FUNCTION_BLOCK FB_SignalTower
VAR_INPUT
    // TRUE: Activates the defined operation
    // FALSE: Aborts/resets the defined operation
    Enable     :BOOL := TRUE;
    LampRed    :REFERENCE TO BOOL;
    LampYellow :REFERENCE TO BOOL;
    LampGreen  :REFERENCE TO BOOL;
    Buzz       :REFERENCE TO BOOL;
	ForceCloseBuzz : BOOL;
	BuzzSwitchOnTime	:LREAL :=3000.0 ; //In Second
END_VAR

VAR_OUTPUT
    // TRUE: Operation is running
    Vaild :BOOL;
    // TRUE: Error condition reached
    Error :BOOL;
    // Error code describing error condition
    ErrorID :DINT;
END_VAR

VAR
    LampRed_Active    :BOOL;         // True :Lamp Red actived
    LampYellow_Active :BOOL;         // True :Lamp Yellow actived
    LampGreen_Active  :BOOL;         // True : Lamp Green actived
    FB_1Hz            :FB_SignalGen; // 1Hz flash signal generator
    FB_2Hz            :FB_SignalGen; // 2Hz flash signal generator
    FB_05Hz           :FB_SignalGen; // 0.5 Hz flash signal generator
    // Signal Tower controller output
    LampSingal :ST_SignalTower;
	BuzzOnTimer			:TON;

END_VAR

// Call Signal generator
A_SignalGenerator();

// 
IF Enable THEN
	LampSingal.Lamp_Red 	:= M_LampRed();
	LampSingal.Lamp_Yellow	:= M_LampYellow();
	LampSingal.Lamp_Green 	:= M_LampGreen();
	LampSingal.Buzz			:=M_Buzz(BuzzSwitchOnTime);
ELSE
	LampSingal.Lamp_Red := FALSE;
	LampSingal.Lamp_Yellow := FALSE;
	LampSingal.Lamp_Green := FALSE;
	LampSingal.Buzz := FALSE;
END_IF

LampRed := LampSingal.Lamp_Red;
LampYellow := LampSingal.Lamp_Yellow;
LampGreen := LampSingal.Lamp_Green;
Buzz := LampSingal.Buzz;

ACTION A_SignalGenerator:
FB_1Hz(PT := F_FtoPT(Hz := 1));
FB_2Hz(PT := F_FtoPT(Hz := 2));
FB_05Hz(PT := F_FtoPT(Hz := 0.5));
END_ACTION

METHOD M_Buzz : BOOL
VAR_INPUT
	SwitchOnTime : LREAL ;//In second
END_VAR
VAR
	SignalMode: E_SignalTowerLampMode:=E_SignalTowerLampMode.Disable;
	
END_VAR
BuzzOnTimer(PT:= DWORD_TO_TIME(LREAL_TO_DWORD(SwitchOnTime*1000)));

IF ForceCloseBuzz THEN
	SignalMode := E_SignalTowerLampMode.Disable;
ELSE
	IF  GVL_ADS.MachineState = E_MachineState.Error THEN
		BuzzOnTimer.IN :=TRUE;		
		SignalMode := E_SignalTowerLampMode.Flash_2Hz;			
	ELSE   
		BuzzOnTimer.IN :=FALSE;
	END_IF
	
END_IF
// Determine the Lamp mode based on the current SignalTowerMode. 
CASE SignalMode OF
    E_SignalTowerLampMode.Disable: // Lamp off
        M_Buzz := FALSE;
    E_SignalTowerLampMode.AlwaysOn: // Lamp on
        M_Buzz := TRUE AND NOT BuzzOnTimer.Q;
    E_SignalTowerLampMode.Flash_05Hz: // Lamp flash 0.25s on 0.25s off
        M_Buzz := FB_05Hz.Q AND NOT BuzzOnTimer.Q;
    E_SignalTowerLampMode.Flash_1Hz: // Lamp flash 0.5s on 0.5s off	
        M_Buzz := FB_1Hz.Q AND NOT BuzzOnTimer.Q ;
    E_SignalTowerLampMode.Flash_2Hz: // Lamp flash 1s on 1s off
        M_Buzz := FB_2Hz.Q AND ( NOT BuzzOnTimer.Q);
END_CASE
END_METHOD

METHOD M_LampGreen : BOOL
VAR_INPUT
END_VAR
VAR
	SignalMode: E_SignalTowerLampMode:=E_SignalTowerLampMode.Disable;
END_VAR
IF NOT LampRed_Active  THEN
    IF GVL_ADS.MachineState=E_MachineState.Running THEN
        SignalMode := E_SignalTowerLampMode.AlwaysOn;
    ELSE
        SignalMode := E_SignalTowerLampMode.Disable;
    END_IF
ELSIF LampRed_Active  THEN
    SignalMode := E_SignalTowerLampMode.Disable;
END_IF;

// Determine the Lamp mode based on the current SignalTowerMode. 
CASE SignalMode OF
    E_SignalTowerLampMode.Disable: // Lamp off
        M_LampGreen := FALSE;
    E_SignalTowerLampMode.AlwaysOn: // Lamp on
        M_LampGreen := TRUE;
    E_SignalTowerLampMode.Flash_05Hz: // Lamp flash 0.25s on 0.25s off
        M_LampGreen := FB_05Hz.Q;
    E_SignalTowerLampMode.Flash_1Hz: // Lamp flash 0.5s on 0.5s off	
        M_LampGreen := FB_1Hz.Q;
    E_SignalTowerLampMode.Flash_2Hz: // Lamp flash 1s on 1s off
        M_LampGreen := FB_2Hz.Q;
END_CASE

// Lamp effective flag
IF SignalMode = E_SignalTowerLampMode.Disable THEN
    LampGreen_Active := FALSE;
ELSE
    LampGreen_Active := TRUE;
END_IF
END_METHOD

METHOD M_LampRed : BOOL
VAR_INPUT
END_VAR
VAR
	SignalMode: E_SignalTowerLampMode:=E_SignalTowerLampMode.Disable;
END_VAR
// Control SignalMode here
IF GVL_ADS.MachineState=E_MachineState.Error THEN
	SignalMode := E_SignalTowerLampMode.Flash_1Hz;
ELSIF GVL_ADS.MachineState=E_MachineState.StandBy THEN
	SignalMode := E_SignalTowerLampMode.AlwaysOn;	
ELSE
	SignalMode := E_SignalTowerLampMode.Disable;
END_IF
// Determine the Lamp mode based on the current SignalTowerMode. 
CASE SignalMode OF
    E_SignalTowerLampMode.Disable: // Lamp off
        M_LampRed := FALSE;
    E_SignalTowerLampMode.AlwaysOn:// Lamp on
        M_LampRed := TRUE;
    E_SignalTowerLampMode.Flash_05Hz:// Lamp flash 0.25s on 0.25s off
        M_LampRed := FB_05Hz.Q;
    E_SignalTowerLampMode.Flash_1Hz: // Lamp flash 0.5s on 0.5s off
        M_LampRed := FB_1Hz.Q;
    E_SignalTowerLampMode.Flash_2Hz: // Lamp flash 1s on 1s off
        M_LampRed := FB_2Hz.Q;
END_CASE
// Lamp effective flag
IF SignalMode = E_SignalTowerLampMode.Disable THEN
	LampRed_Active := FALSE;
ELSE
	LampRed_Active := TRUE;
END_IF
END_METHOD

METHOD M_LampYellow : BOOL
VAR_INPUT
END_VAR
VAR
	SignalMode: E_SignalTowerLampMode:=E_SignalTowerLampMode.Disable;
END_VAR
// Contorl Signal here
 IF GVL_ADS.MachineState=E_MachineState.NotHomed OR GVL_ADS.MachineState=E_MachineState.Homing THEN
	
		SignalMode := E_SignalTowerLampMode.Flash_2Hz;
	ELSIF GVL_ADS.MachineState=E_MachineState.Homed THEN
		SignalMode := E_SignalTowerLampMode.AlwaysOn;
	ELSE	
		SignalMode := E_SignalTowerLampMode.Disable;
	
END_IF

// Determine the Lamp mode based on the current SignalTowerMode. 
CASE SignalMode OF
    E_SignalTowerLampMode.Disable: // Lamp off
        M_LampYellow := FALSE;
    E_SignalTowerLampMode.AlwaysOn:// Lamp on
        M_LampYellow := TRUE;
    E_SignalTowerLampMode.Flash_05Hz:// Lamp flash 0.25s on 0.25s off
        M_LampYellow := FB_05Hz.Q;
    E_SignalTowerLampMode.Flash_1Hz: // Lamp flash 0.5s on 0.5s off
        M_LampYellow := FB_1Hz.Q;
    E_SignalTowerLampMode.Flash_2Hz: // Lamp flash 1s on 1s off
        M_LampYellow := FB_2Hz.Q;
END_CASE
// Lamp effective flag
IF SignalMode = E_SignalTowerLampMode.Disable THEN
	LampYellow_Active := FALSE;
ELSE
	LampYellow_Active := TRUE;
END_IF
END_METHOD

PROPERTY PUBLIC P_LampGreenState : Bool
GET
P_LampGreenState:=LampSingal.Lamp_Green ;
END_GET
END_PROPERTY

PROPERTY PUBLIC P_LampRedState : Bool
GET
P_LampRedState:=LampSingal.Lamp_Red ;
END_GET
END_PROPERTY

PROPERTY PUBLIC P_LampYellowState : Bool
GET
P_LampYellowState:=LampSingal.Lamp_Yellow ;
END_GET
END_PROPERTY

END_FUNCTION_BLOCK

(* stored: Version 1.1.0.1, ProductVersion 3.1.4024.13
   POU FB_SignalTower: Id {1dc42b3a-9534-40d3-bab1-9a3fd3352017}, SpecialFunc None
   Action A_SignalGenerator: Id {5007de43-27f1-4df8-92e2-4501fa1e4fb4}
   Method M_Buzz: Id {eff69fa8-3ec3-47de-a0a3-b9a78f3ee27f}
   Method M_LampGreen: Id {a34f9e17-3182-4649-a7d4-28e8815d4d82}
   Method M_LampRed: Id {2329bb26-8597-4c80-ba05-709f9c456d84}
   Method M_LampYellow: Id {0bcbdcd0-592a-44c7-8516-36ee953c07fb}
   Property P_LampGreenState: Id {001bb7d5-fcd9-49d5-b915-4c7352c9f451}
   Get Get: Id {7872edae-3f10-4cb4-8814-41f53fdcb548}
   Property P_LampRedState: Id {82e88a37-2ba5-4ccb-abee-319e5534e2a0}
   Get Get: Id {0bf4bbec-7894-4a3f-9a31-740f2e5d75fc}
   Property P_LampYellowState: Id {8bdb4f40-3f1d-4b5f-8d18-0ef7118a9ade}
   Get Get: Id {1938b688-657c-4021-8520-6d4c24a0d84d} *)
